// TIA Portal project "FillerMachine" (V15)
// Maquina llenadora Fuente Pura CCN

(* hardware
DEVICE "ET 200SP station_1"  ET 200SP-Station
   slot 0: "Rack_0"  Rack  6ES5 710-8MAx1
   slot 1: "PLC_1"  CPU 1510SP-1 PN  6ES7 510-1DJ01-0AB0  V2.5
   slot 2: "DI 8x24VDC ST_1"  DI 8x24VDC ST  6ES7 131-6BF00-0BA0  V1.1
      slot 1: "DI 8x24VDC ST_1"  DI 8x24VDC ST
   slot 3: "DI 8x24VDC ST_2"  DI 8x24VDC ST  6ES7 131-6BF01-0BA0  V0.0
      slot 1: "DI 8x24VDC ST_2"  DI 8x24VDC ST
   slot 4: "DI 8x24VDC ST_3"  DI 8x24VDC ST  6ES7 131-6BF01-0BA0  V0.0
      slot 1: "DI 8x24VDC ST_3"  DI 8x24VDC ST
   slot 5: "DQ 8x24VDC/0.5A ST_1"  DQ 8x24VDC/0.5A ST  6ES7 132-6BF01-0BA0  V0.0
      slot 1: "DQ 8x24VDC/0.5A ST_1"  DQ 8x24VDC/0.5A ST
   slot 6: "DQ 8x24VDC/0.5A ST_2"  DQ 8x24VDC/0.5A ST  6ES7 132-6BF01-0BA0  V0.0
      slot 1: "DQ 8x24VDC/0.5A ST_2"  DQ 8x24VDC/0.5A ST
   slot 7: "DQ 8x24VDC/0.5A ST_3"  DQ 8x24VDC/0.5A ST  6ES7 132-6BF01-0BA0  V0.0
      slot 1: "DQ 8x24VDC/0.5A ST_3"  DQ 8x24VDC/0.5A ST
   slot 8: "Server module_1"  Server module  6ES7 193-6PA00-0AA0  V1.1
      slot 1: "Server module_1"  Server module
   slot 127: "BA 2xRJ45"  BA 2xRJ45  6ES7 193-6AR00-0AA0  V0.0
      slot 32769: "Port_1"  6ES7 193-6AR00-0AA0
      slot 32770: "Port_2"  6ES7 193-6AR00-0AA0
DEVICE "HMI_1"  KTP600 Basic color PN
   slot 0: "HMI_1"  KTP600 Basic color PN  6AV6 647-0AD11-3AX0  12.0.0.0
   slot 1: "HMI_RT_2"  KTP600 Basic color PN  6AV6 647-0AD11-3AX0  12.0.0.0
   slot 5: "HMI_1.IE_CP_1"  PROFINET Interface  12.0.0.0
      slot 1: "PROFINET Interface_1"  PROFINET Interface
         slot 1: "Port_1"  Port
*)

// ===== PLC "PLC_1"  CPU 1510SP-1 PN =====

VAR_GLOBAL   // PLC tag table "Default tag table"
   "Stop_bitin" AT %I2.2 : Bool;
   "TriggerPump" AT %I0.1 : Bool;
   "ACKPump" AT %I0.2 : Bool;
   "TriggerClamp" AT %I0.3 : Bool;
   "ACKClamp" AT %I0.4 : Bool;
   "TriggerTransp1" AT %I0.5 : Bool;
   "ACKTransp1" AT %I0.6 : Bool;
   "TriggerTransp2" AT %I0.7 : Bool;
   "ACKTransp2" AT %I1.0 : Bool;
   "SensorTransIN2" AT %I1.1 : Bool;
   "SensorInBottle" AT %I1.2 : Bool;
   "SensorOutBottle" AT %I1.3 : Bool;
   "SensorLastBottle" AT %I1.4 : Bool;
   "SensorStageIN1" AT %I1.5 : Bool;
   "SensorLevelH" AT %I1.6 : Bool;
   "SensorLevelL" AT %I1.7 : Bool;
   "SensorBottleClamp" AT %I2.0 : Bool;
   "SensorTranspClamp" AT %I2.1 : Bool;
   "PumpVLow" AT %Q0.0 : Bool;
   "PumpVHigh" AT %Q0.1 : Bool;
   "PumpStop" AT %Q0.2 : Bool;
   "MotorTap" AT %Q0.3 : Bool;
   "MotorTrans1" AT %Q0.4 : Bool;
   "MotorTrans2" AT %Q0.5 : Bool;
   "EVPrincip" AT %Q0.6 : Bool;
   "EVBlowCylindIN" AT %Q0.7 : Bool;
   "EVCylindBottleHigh" AT %Q1.6 : Bool;
   "EVCylindNeck" AT %Q1.7 : Bool;
   "EVDoorIn" AT %Q2.2 : Bool;
   "EVDoorOut" AT %Q2.3 : Bool;
   "EVClampBotNeck" AT %Q2.4 : Bool;
   "EVClampDoor" AT %Q2.5 : Bool;
   "EVSuperClamp" AT %Q2.6 : Bool;
   "EVMandrilcylindUpDown" AT %Q2.7 : Bool;
   "MStartTouch" AT %M11.0 : Bool;
   "MBandaT-On" AT %M10.1 : Bool;
   "MFillScreen" AT %M10.2 : Bool;
   "MBottleProcess" AT %MD100 : DInt;
   "MBottleCounterIN" AT %MD4 : DInt;
   "MBottleCounterOut" AT %MD12 : DInt;
   "MEnableClampValve" AT %MD16 : DInt;
   "MFillFinish" AT %M10.3 : Bool;
   "M_stop_bit" AT %M11.1 : Bool;
   "F_TriggerPump" AT %M11.3 : Bool;
   "F_ACKPump" AT %M11.4 : Bool;
   "F_TriggerClamp" AT %M11.5 : Bool;
   "F_ACKClamp" AT %M11.6 : Bool;
   "F_TriggerTransp1" AT %M11.7 : Bool;
   "F_ACKTransp1" AT %M20.0 : Bool;
   "F_TriggerTransp2" AT %M20.1 : Bool;
   "F_ACKTransp2" AT %M20.2 : Bool;
   "SensorTransIN2_bit" AT %M20.3 : Bool;
   "SensorInBottle_bit" AT %M20.4 : Bool;
   "SensorOutBottle_bit" AT %M20.5 : Bool;
   "SensorLastBottle_bit" AT %M20.6 : Bool;
   "SensorStageIN1_bit" AT %M20.7 : Bool;
   "SensorLevelH_bit" AT %M21.0 : Bool;
   "SensorLevelL_bit" AT %M21.1 : Bool;
   "SensorBottleClamp_bit" AT %M21.2 : Bool;
   "SensorTranspClamp_bit" AT %M21.3 : Bool;
   "PumpVLow_bit" AT %M21.4 : Bool;
   "PumpVHigh_bit" AT %M21.5 : Bool;
   "PumpStop_bit" AT %M21.6 : Bool;
   "MotorTap_bit" AT %M21.7 : Bool;
   "MotorTrans1_bit" AT %M22.0 : Bool;
   "MotorTrans2_bit" AT %M22.1 : Bool;
   "EVPrincip_bit" AT %M22.2 : Bool;
   "EVBlowCylindIN_bit" AT %M22.3 : Bool;
   "EVMandrilcylindUpDown_bit" AT %M22.4 : Bool;
   "EVCylindNeck_bit" AT %M22.5 : Bool;
   "EVDoorIn_bit" AT %M22.6 : Bool;
   "EVDoorOut_bit" AT %M22.7 : Bool;
   "EVClampBotNeck_bit" AT %M23.0 : Bool;
   "EVClampDoor_bit" AT %M23.1 : Bool;
   "EVSuperClamp_bit" AT %M23.2 : Bool;
   "Alarm" AT %M24.0 : Bool;
   "F_TriggerPump_bit" AT %M24.1 : Bool;
   "F_ACKPump_bit" AT %M24.2 : Bool;
   "F_TriggerClamp_bit" AT %M24.3 : Bool;
   "F_ACKClamp_bit" AT %M24.4 : Bool;
   "F_TriggerTransp1_bit" AT %M24.5 : Bool;
   "F_ACKTransp1_bit" AT %M24.6 : Bool;
   "F_TriggerTransp2_bit" AT %M24.7 : Bool;
   "F_ACKTransp2_bit" AT %M25.0 : Bool;
   "Run" AT %M25.1 : Bool;
   "Stop_bit" AT %M25.2 : Bool;
   "StageLL0" AT %M25.3 : Bool;
   "StageLL1" AT %M25.4 : Bool;
   "MBottleCounterR" AT %M25.5 : Bool;
   "MBottleProcessR" AT %M25.6 : Bool;
   "StageLL2" AT %M25.7 : Bool;
   "MBottleclampRt" AT %M27.3 : Bool;
   "MBottleClamProcess" AT %MD101 : DInt;
   "MTrans1_touch" AT %M27.4 : Bool;
   "MTrans2_touch" AT %M27.5 : Bool;
   "MPump_touch" AT %M27.6 : Bool;
   "MClamp_touch" AT %M27.7 : Bool;
   "EVCylindBottleHigh_bit" AT %M28.0 : Bool;
   "StageLL3" AT %M28.1 : Bool;
   "StageLL4" AT %M28.2 : Bool;
   "StageLL5" AT %M28.3 : Bool;
   "StageLL6" AT %M28.4 : Bool;
   "StageLL7" AT %M28.5 : Bool;
   "StageLL8" AT %M28.6 : Bool;
   "StageLL9" AT %M28.7 : Bool;
   "StageLL10" AT %M29.0 : Bool;
   "StageLL11" AT %M29.1 : Bool;
   "Tag_1" AT %M400.1 : Bool;
   "StageLL12" AT %M29.2 : Bool;
   "StageLL13" AT %M29.3 : Bool;
   "StageLL14" AT %M29.4 : Bool;
   "Tag_2" AT %M400.2 : Bool;
   "StageLL00" AT %M29.5 : Bool;
   "MBottleCounterOutR" AT %M29.6 : Bool;
   "StageTap0" AT %M29.7 : Bool;
   "StageTap1" AT %M30.0 : Bool;
   "StageTap2" AT %M30.1 : Bool;
   "StageTap3" AT %M30.2 : Bool;
   "StageTap4" AT %M30.3 : Bool;
   "StageTap5" AT %M30.4 : Bool;
   "MTapProcessR" AT %M30.5 : Bool;
   "StageCon0" AT %M30.6 : Bool;
   "StageCon1" AT %M30.7 : Bool;
   "StageCon2" AT %M31.0 : Bool;
   "StageCon3" AT %M31.1 : Bool;
   "MConvT1R" AT %M31.2 : Bool;
   "MConvT2R" AT %M31.3 : Bool;
END_VAR

DATA_BLOCK "DB_Alarms"   // DB13
{ S7_Optimized_Access := 'FALSE' }
VERSION : 0.1
   VAR
      Stop_alm : Bool;
      T_Pump_alm : Bool;
      T_Transp1_alm : Bool;
      T_Transp2_alm : Bool;
      T_Clamp_alm_1 : Bool;
      alarms_active : Bool;
   END_VAR
BEGIN
END_DATA_BLOCK

// folder: System blocks/Program resources

DATA_BLOCK "IEC_Counter_0_DB"   // DB1
{ S7_Optimized_Access := 'TRUE' }
AUTHOR : Simatic
FAMILY : IEC
NAME : CNTR
VERSION : 1.0
// stored: InstanceOfName IEC_COUNTER
"IEC_COUNTER"
BEGIN
END_DATA_BLOCK

DATA_BLOCK "IEC_Timer_0_DB"   // DB2
{ S7_Optimized_Access := 'TRUE' }
AUTHOR : Simatic
FAMILY : IEC
NAME : IEC_TMR
VERSION : 1.0
// stored: InstanceOfName IEC_TIMER
"IEC_TIMER"
BEGIN
END_DATA_BLOCK

DATA_BLOCK "IEC_Timer_0_DB_1"   // DB3
{ S7_Optimized_Access := 'TRUE' }
AUTHOR : Simatic
FAMILY : IEC
NAME : IEC_TMR
VERSION : 1.0
// stored: InstanceOfName IEC_TIMER
"IEC_TIMER"
BEGIN
END_DATA_BLOCK

DATA_BLOCK "IEC_Timer_0_DB_2"   // DB5
{ S7_Optimized_Access := 'TRUE' }
AUTHOR : Simatic
FAMILY : IEC
NAME : IEC_TMR
VERSION : 1.0
// stored: InstanceOfName IEC_TIMER
"IEC_TIMER"
BEGIN
END_DATA_BLOCK

DATA_BLOCK "IEC_Timer_0_DB_4"   // DB6
{ S7_Optimized_Access := 'TRUE' }
AUTHOR : Simatic
FAMILY : IEC
NAME : IEC_TMR
VERSION : 1.0
// stored: InstanceOfName IEC_TIMER
"IEC_TIMER"
BEGIN
END_DATA_BLOCK

DATA_BLOCK "IEC_Timer_0_DB_5"   // DB7
{ S7_Optimized_Access := 'TRUE' }
AUTHOR : Simatic
FAMILY : IEC
NAME : IEC_TMR
VERSION : 1.0
// stored: InstanceOfName IEC_TIMER
"IEC_TIMER"
BEGIN
END_DATA_BLOCK

DATA_BLOCK "IEC_Timer_0_DB_17"   // DB8
{ S7_Optimized_Access := 'TRUE' }
AUTHOR : Simatic
FAMILY : IEC
NAME : IEC_TMR
VERSION : 1.0
// stored: InstanceOfName IEC_TIMER
"IEC_TIMER"
BEGIN
END_DATA_BLOCK

DATA_BLOCK "IEC_Timer_0_DB_7"   // DB9
{ S7_Optimized_Access := 'TRUE' }
AUTHOR : Simatic
FAMILY : IEC
NAME : IEC_TMR
VERSION : 1.0
// stored: InstanceOfName IEC_TIMER
"IEC_TIMER"
BEGIN
END_DATA_BLOCK

DATA_BLOCK "IEC_Timer_0_DB_8"   // DB10
{ S7_Optimized_Access := 'TRUE' }
AUTHOR : Simatic
FAMILY : IEC
NAME : IEC_TMR
VERSION : 1.0
// stored: InstanceOfName IEC_TIMER
"IEC_TIMER"
BEGIN
END_DATA_BLOCK

DATA_BLOCK "IEC_Timer_0_DB_9"   // DB11
{ S7_Optimized_Access := 'TRUE' }
AUTHOR : Simatic
FAMILY : IEC
NAME : IEC_TMR
VERSION : 1.0
// stored: InstanceOfName IEC_TIMER
"IEC_TIMER"
BEGIN
END_DATA_BLOCK

DATA_BLOCK "IEC_Timer_0_DB_10"   // DB12
{ S7_Optimized_Access := 'TRUE' }
AUTHOR : Simatic
FAMILY : IEC
NAME : IEC_TMR
VERSION : 1.0
// stored: InstanceOfName IEC_TIMER
"IEC_TIMER"
BEGIN
END_DATA_BLOCK

DATA_BLOCK "IEC_Counter_1_DB"   // DB14
{ S7_Optimized_Access := 'TRUE' }
AUTHOR : Simatic
FAMILY : IEC
NAME : CNTR
VERSION : 1.0
// stored: InstanceOfName IEC_COUNTER
"IEC_COUNTER"
BEGIN
END_DATA_BLOCK

DATA_BLOCK "IEC_Timer_0_DB_11"   // DB15
{ S7_Optimized_Access := 'TRUE' }
AUTHOR : Simatic
FAMILY : IEC
NAME : IEC_TMR
VERSION : 1.0
// stored: InstanceOfName IEC_TIMER
"IEC_TIMER"
BEGIN
END_DATA_BLOCK

DATA_BLOCK "IEC_Timer_0_DB_12"   // DB16
{ S7_Optimized_Access := 'TRUE' }
AUTHOR : Simatic
FAMILY : IEC
NAME : IEC_TMR
VERSION : 1.0
// stored: InstanceOfName IEC_TIMER
"IEC_TIMER"
BEGIN
END_DATA_BLOCK

DATA_BLOCK "IEC_Timer_0_DB_13"   // DB17
{ S7_Optimized_Access := 'TRUE' }
AUTHOR : Simatic
FAMILY : IEC
NAME : IEC_TMR
VERSION : 1.0
// stored: InstanceOfName IEC_TIMER
"IEC_TIMER"
BEGIN
END_DATA_BLOCK

DATA_BLOCK "IEC_Timer_0_DB_14"   // DB18
{ S7_Optimized_Access := 'TRUE' }
AUTHOR : Simatic
FAMILY : IEC
NAME : IEC_TMR
VERSION : 1.0
// stored: InstanceOfName IEC_TIMER
"IEC_TIMER"
BEGIN
END_DATA_BLOCK

DATA_BLOCK "IEC_Timer_0_DB_15"   // DB19
{ S7_Optimized_Access := 'TRUE' }
AUTHOR : Simatic
FAMILY : IEC
NAME : IEC_TMR
VERSION : 1.0
// stored: InstanceOfName IEC_TIMER
"IEC_TIMER"
BEGIN
END_DATA_BLOCK

DATA_BLOCK "IEC_Timer_0_DB_16"   // DB20
{ S7_Optimized_Access := 'TRUE' }
AUTHOR : Simatic
FAMILY : IEC
NAME : IEC_TMR
VERSION : 1.0
// stored: InstanceOfName IEC_TIMER
"IEC_TIMER"
BEGIN
END_DATA_BLOCK

// folder: (top level)

ORGANIZATION_BLOCK "Main"   // OB1, LAD, ProgramCycle
TITLE = "Main Program Sweep (Cycle)"
{ S7_Optimized_Access := 'TRUE' }
VERSION : 0.1
   VAR_INPUT
      Initial_Call : Bool;   // Initial call of this OB
      Remanence : Bool;   // =True, if remanent data are available
   END_VAR
   VAR_TEMP   // added for the SCL form of the ladder/FBD networks
      _w1 : Bool;
   END_VAR
BEGIN

REGION Network 1
   // Start  Stop Control
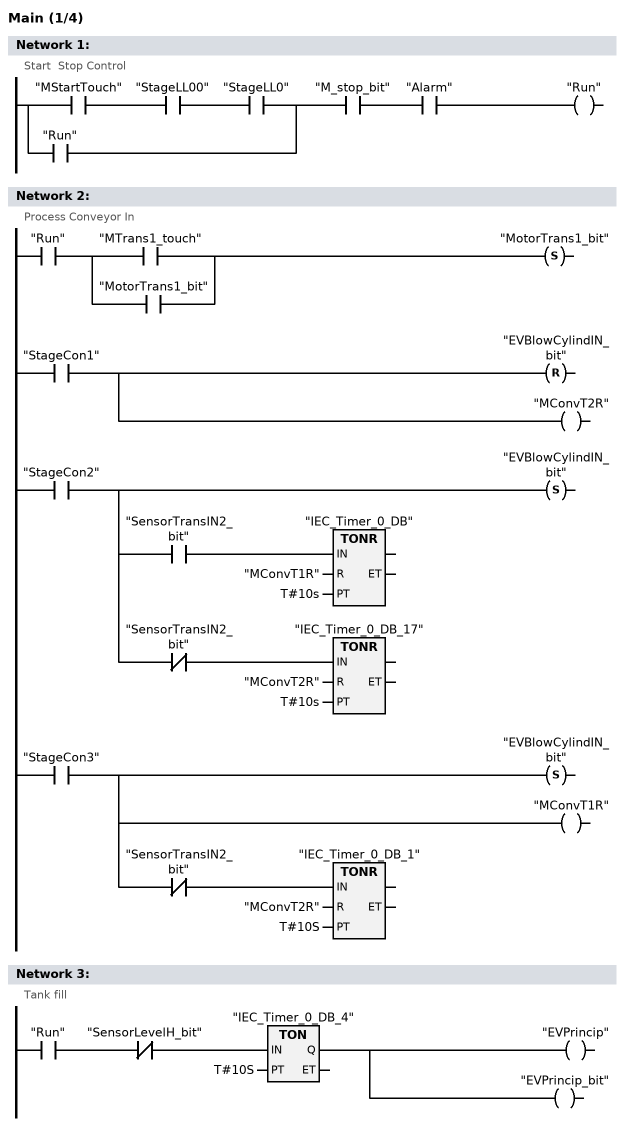
   RUNG wire#powerrail
      Contact( "MStartTouch" )
      Contact( "StageLL00" )
      Contact( "StageLL0" )
      wire#w1
      Contact( "M_stop_bit" )
      Contact( "Alarm" )
      Coil( "Run" )
   END_RUNG
   RUNG wire#powerrail
      Contact( "Run" )
   END_RUNG wire#w1
   // the same network as SCL:
   "Run" := (("MStartTouch" AND "StageLL00" AND "StageLL0") OR "Run") AND "M_stop_bit" AND "Alarm";
END_REGION

REGION Network 2
   // Process Conveyor In
   IF "Run" AND ("MTrans1_touch" OR "MotorTrans1_bit") THEN "MotorTrans1_bit" := TRUE; END_IF;
   IF "StageCon1" THEN "EVBlowCylindIN_bit" := FALSE; END_IF;
   "MConvT2R" := "StageCon1";
   IF "StageCon2" THEN "EVBlowCylindIN_bit" := TRUE; END_IF;
   "IEC_Timer_0_DB".TONR(IN := "StageCon2" AND "SensorTransIN2_bit", R := "MConvT1R", PT := T#10s);
   "IEC_Timer_0_DB_17".TONR(IN := "StageCon2" AND NOT "SensorTransIN2_bit", R := "MConvT2R", PT := T#10s);
   IF "StageCon3" THEN "EVBlowCylindIN_bit" := TRUE; END_IF;
   "MConvT1R" := "StageCon3";
   "IEC_Timer_0_DB_1".TONR(IN := "StageCon3" AND NOT "SensorTransIN2_bit", R := "MConvT2R", PT := T#10S);
END_REGION

REGION Network 3
   // Tank fill
   "IEC_Timer_0_DB_4".TON(IN := "Run" AND NOT "SensorLevelH_bit", PT := T#10S);
   "EVPrincip" := "IEC_Timer_0_DB_4".Q;
   "EVPrincip_bit" := "IEC_Timer_0_DB_4".Q;
END_REGION

REGION Network 4
   // Process Filling Bottle
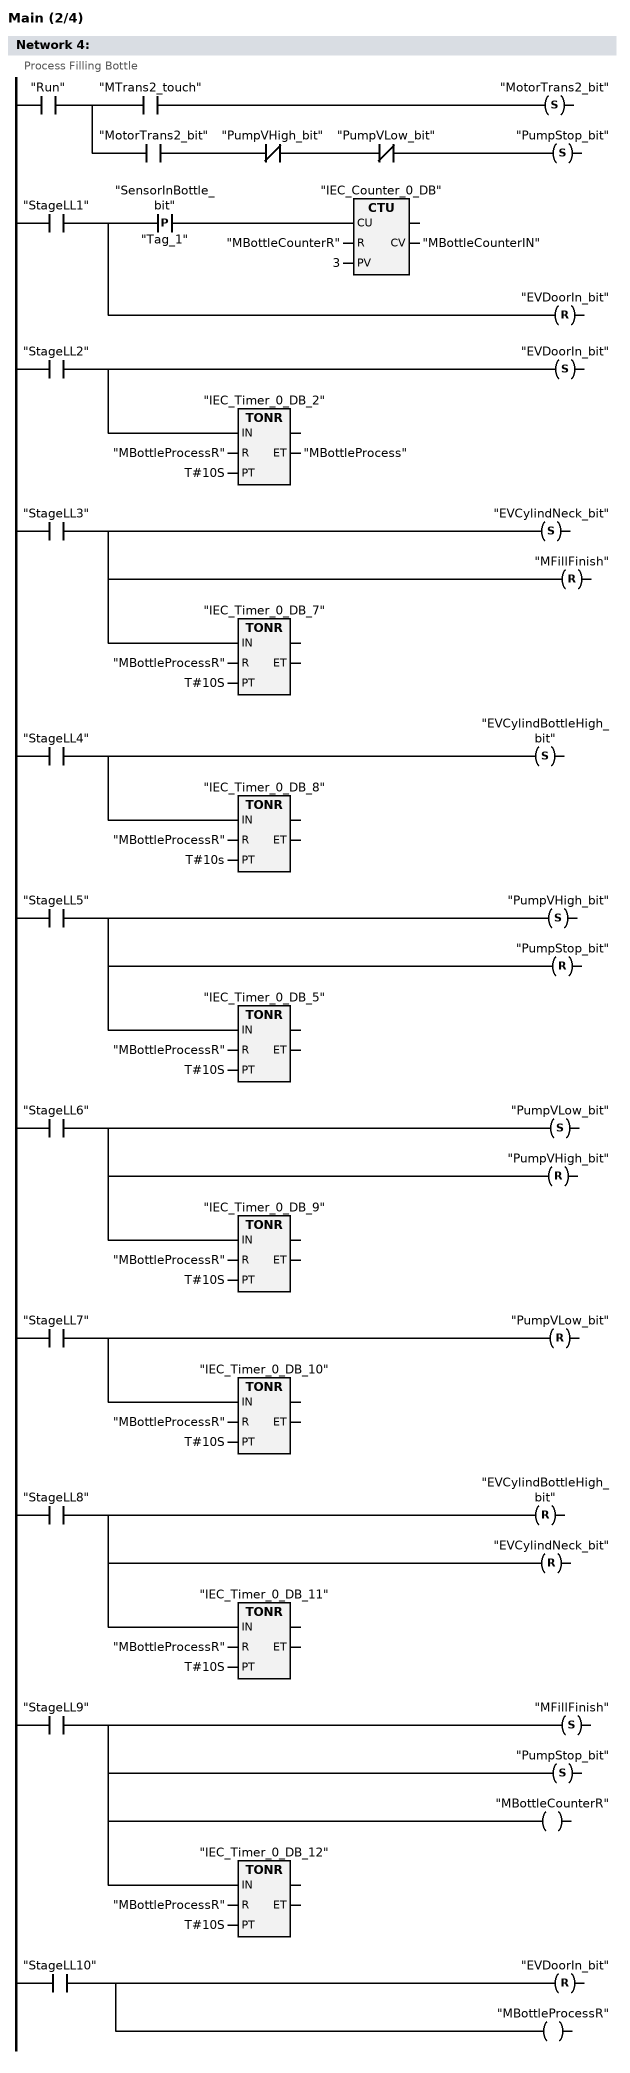
   IF "Run" AND "MTrans2_touch" THEN "MotorTrans2_bit" := TRUE; END_IF;
   IF "Run" AND "MotorTrans2_bit" AND NOT "PumpVHigh_bit" AND NOT "PumpVLow_bit" THEN
       "PumpStop_bit" := TRUE;
   END_IF;
   #_w1 := "StageLL1" AND "SensorInBottle_bit" AND NOT "Tag_1";   // rising edge of "SensorInBottle_bit"
   "Tag_1" := "SensorInBottle_bit";
   "IEC_Counter_0_DB".CTU(CU := #_w1, R := "MBottleCounterR", PV := 3, CV => "MBottleCounterIN");
   IF "StageLL1" THEN "EVDoorIn_bit" := FALSE; END_IF;
   IF "StageLL2" THEN "EVDoorIn_bit" := TRUE; END_IF;
   "IEC_Timer_0_DB_2".TONR(IN := "StageLL2", R := "MBottleProcessR", PT := T#10S, ET => "MBottleProcess");
   IF "StageLL3" THEN
       "EVCylindNeck_bit" := TRUE;
       "MFillFinish" := FALSE;
   END_IF;
   "IEC_Timer_0_DB_7".TONR(IN := "StageLL3", R := "MBottleProcessR", PT := T#10S);
   IF "StageLL4" THEN "EVCylindBottleHigh_bit" := TRUE; END_IF;
   "IEC_Timer_0_DB_8".TONR(IN := "StageLL4", R := "MBottleProcessR", PT := T#10s);
   IF "StageLL5" THEN
       "PumpVHigh_bit" := TRUE;
       "PumpStop_bit" := FALSE;
   END_IF;
   "IEC_Timer_0_DB_5".TONR(IN := "StageLL5", R := "MBottleProcessR", PT := T#10S);
   IF "StageLL6" THEN
       "PumpVLow_bit" := TRUE;
       "PumpVHigh_bit" := FALSE;
   END_IF;
   "IEC_Timer_0_DB_9".TONR(IN := "StageLL6", R := "MBottleProcessR", PT := T#10S);
   IF "StageLL7" THEN "PumpVLow_bit" := FALSE; END_IF;
   "IEC_Timer_0_DB_10".TONR(IN := "StageLL7", R := "MBottleProcessR", PT := T#10S);
   IF "StageLL8" THEN
       "EVCylindBottleHigh_bit" := FALSE;
       "EVCylindNeck_bit" := FALSE;
   END_IF;
   "IEC_Timer_0_DB_11".TONR(IN := "StageLL8", R := "MBottleProcessR", PT := T#10S);
   IF "StageLL9" THEN
       "MFillFinish" := TRUE;
       "PumpStop_bit" := TRUE;
   END_IF;
   "MBottleCounterR" := "StageLL9";
   "IEC_Timer_0_DB_12".TONR(IN := "StageLL9", R := "MBottleProcessR", PT := T#10S);
   IF "StageLL10" THEN "EVDoorIn_bit" := FALSE; END_IF;
   "MBottleProcessR" := "StageLL10";
END_REGION

REGION Network 5
   // Cylindre out
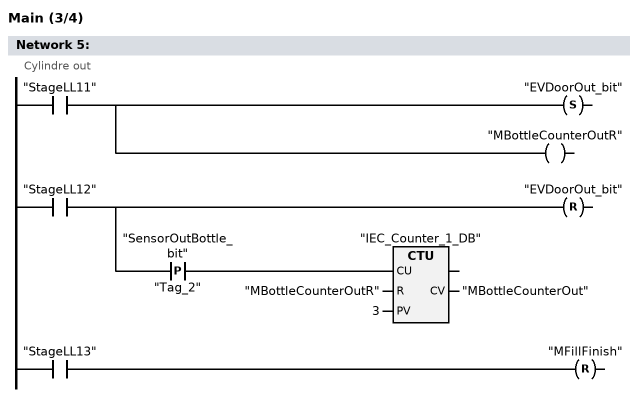
   IF "StageLL11" THEN "EVDoorOut_bit" := TRUE; END_IF;
   "MBottleCounterOutR" := "StageLL11";
   IF "StageLL12" THEN "EVDoorOut_bit" := FALSE; END_IF;
   #_w1 := "StageLL12" AND "SensorOutBottle_bit" AND NOT "Tag_2";   // rising edge of "SensorOutBottle_bit"
   "Tag_2" := "SensorOutBottle_bit";
   "IEC_Counter_1_DB".CTU(CU := #_w1, R := "MBottleCounterOutR", PV := 3, CV => "MBottleCounterOut");
   IF "StageLL13" THEN "MFillFinish" := FALSE; END_IF;
END_REGION

REGION Network 6
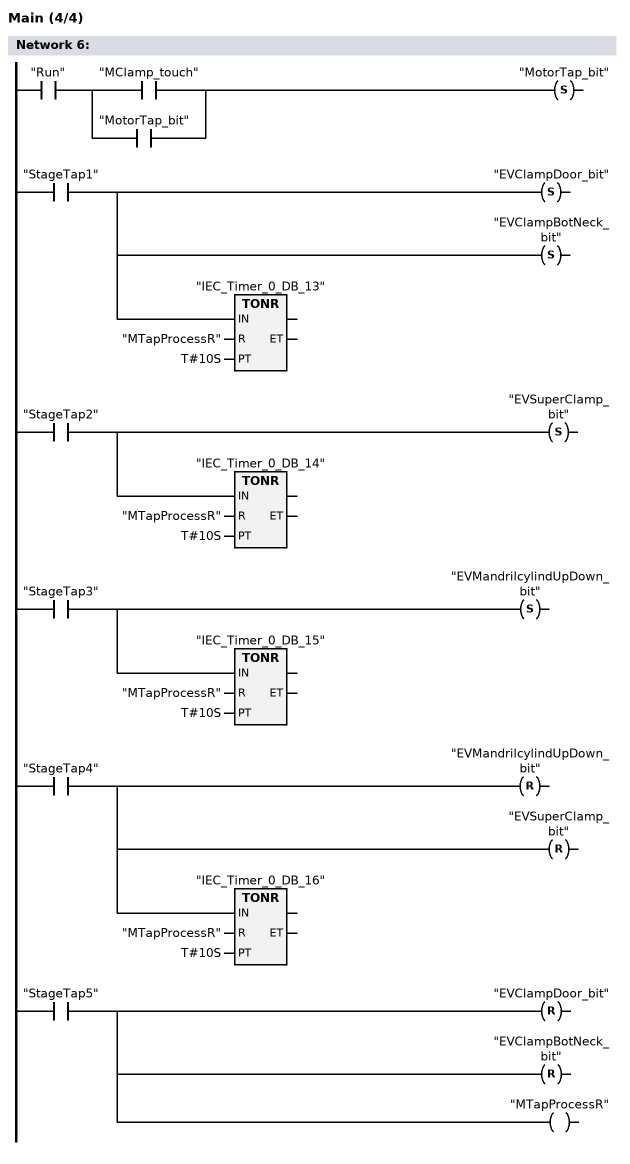
   IF "Run" AND ("MClamp_touch" OR "MotorTap_bit") THEN "MotorTap_bit" := TRUE; END_IF;
   IF "StageTap1" THEN
       "EVClampDoor_bit" := TRUE;
       "EVClampBotNeck_bit" := TRUE;
   END_IF;
   "IEC_Timer_0_DB_13".TONR(IN := "StageTap1", R := "MTapProcessR", PT := T#10S);
   IF "StageTap2" THEN "EVSuperClamp_bit" := TRUE; END_IF;
   "IEC_Timer_0_DB_14".TONR(IN := "StageTap2", R := "MTapProcessR", PT := T#10S);
   IF "StageTap3" THEN "EVMandrilcylindUpDown_bit" := TRUE; END_IF;
   "IEC_Timer_0_DB_15".TONR(IN := "StageTap3", R := "MTapProcessR", PT := T#10S);
   IF "StageTap4" THEN
       "EVMandrilcylindUpDown_bit" := FALSE;
       "EVSuperClamp_bit" := FALSE;
   END_IF;
   "IEC_Timer_0_DB_16".TONR(IN := "StageTap4", R := "MTapProcessR", PT := T#10S);
   IF "StageTap5" THEN
       "EVClampDoor_bit" := FALSE;
       "EVClampBotNeck_bit" := FALSE;
   END_IF;
   "MTapProcessR" := "StageTap5";
END_REGION

REGION Network 7
   // Minor bits
END_REGION
END_ORGANIZATION_BLOCK

ORGANIZATION_BLOCK "Alarms_block"   // OB123, LAD, ProgramCycle
TITLE = "Main Program Sweep (Cycle)"
{ S7_Optimized_Access := 'TRUE' }
VERSION : 0.1
   VAR_INPUT
      Initial_Call : Bool;   // Initial call of this OB
      Remanence : Bool;   // =True, if remanent data are available
   END_VAR
BEGIN

REGION Network 1
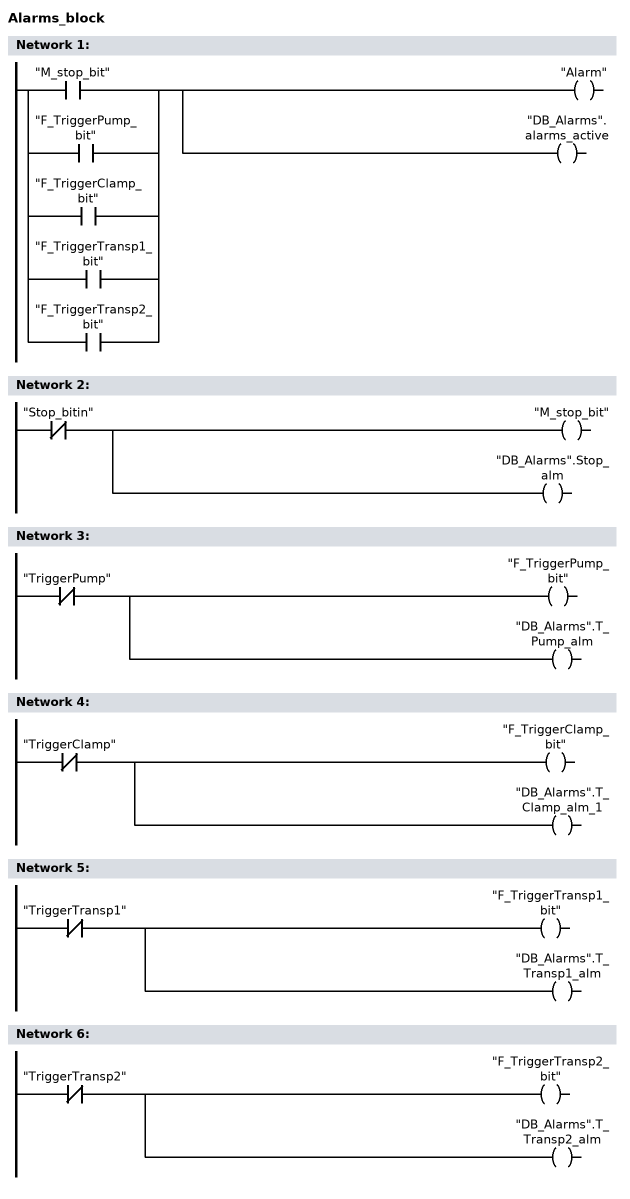
   RUNG wire#powerrail
      Contact( "M_stop_bit" )
      wire#w1
      Coil( "Alarm" )
   END_RUNG
   RUNG wire#powerrail
      Contact( "F_TriggerPump_bit" )
   END_RUNG wire#w1
   RUNG wire#powerrail
      Contact( "F_TriggerClamp_bit" )
   END_RUNG wire#w1
   RUNG wire#powerrail
      Contact( "F_TriggerTransp1_bit" )
   END_RUNG wire#w1
   RUNG wire#powerrail
      Contact( "F_TriggerTransp2_bit" )
   END_RUNG wire#w1
   RUNG wire#w1
      Coil( "DB_Alarms".alarms_active )
   END_RUNG
   // the same network as SCL:
   "Alarm" := "M_stop_bit" OR "F_TriggerPump_bit" OR "F_TriggerClamp_bit" OR "F_TriggerTransp1_bit" OR "F_TriggerTransp2_bit";
   "DB_Alarms".alarms_active := "Alarm";
END_REGION

REGION Network 2
   RUNG wire#powerrail
      I_Contact( "Stop_bitin" )
      wire#w1
      Coil( "M_stop_bit" )
   END_RUNG
   RUNG wire#w1
      Coil( "DB_Alarms".Stop_alm )
   END_RUNG
   // the same network as SCL:
   "M_stop_bit" := NOT "Stop_bitin";
   "DB_Alarms".Stop_alm := NOT "Stop_bitin";
END_REGION

REGION Network 3
   RUNG wire#powerrail
      I_Contact( "TriggerPump" )
      wire#w1
      Coil( "F_TriggerPump_bit" )
   END_RUNG
   RUNG wire#w1
      Coil( "DB_Alarms".T_Pump_alm )
   END_RUNG
   // the same network as SCL:
   "F_TriggerPump_bit" := NOT "TriggerPump";
   "DB_Alarms".T_Pump_alm := NOT "TriggerPump";
END_REGION

REGION Network 4
   RUNG wire#powerrail
      I_Contact( "TriggerClamp" )
      wire#w1
      Coil( "F_TriggerClamp_bit" )
   END_RUNG
   RUNG wire#w1
      Coil( "DB_Alarms".T_Clamp_alm_1 )
   END_RUNG
   // the same network as SCL:
   "F_TriggerClamp_bit" := NOT "TriggerClamp";
   "DB_Alarms".T_Clamp_alm_1 := NOT "TriggerClamp";
END_REGION

REGION Network 5
   RUNG wire#powerrail
      I_Contact( "TriggerTransp1" )
      wire#w1
      Coil( "F_TriggerTransp1_bit" )
   END_RUNG
   RUNG wire#w1
      Coil( "DB_Alarms".T_Transp1_alm )
   END_RUNG
   // the same network as SCL:
   "F_TriggerTransp1_bit" := NOT "TriggerTransp1";
   "DB_Alarms".T_Transp1_alm := NOT "TriggerTransp1";
END_REGION

REGION Network 6
   RUNG wire#powerrail
      I_Contact( "TriggerTransp2" )
      wire#w1
      Coil( "F_TriggerTransp2_bit" )
   END_RUNG
   RUNG wire#w1
      Coil( "DB_Alarms".T_Transp2_alm )
   END_RUNG
   // the same network as SCL:
   "F_TriggerTransp2_bit" := NOT "TriggerTransp2";
   "DB_Alarms".T_Transp2_alm := NOT "TriggerTransp2";
END_REGION
END_ORGANIZATION_BLOCK

ORGANIZATION_BLOCK "Stages"   // OB124, LAD, ProgramCycle
TITLE = "Main Program Sweep (Cycle)"
{ S7_Optimized_Access := 'TRUE' }
VERSION : 0.1
   VAR_INPUT
      Initial_Call : Bool;   // Initial call of this OB
      Remanence : Bool;   // =True, if remanent data are available
   END_VAR
   VAR_TEMP   // added for the SCL form of the ladder/FBD networks
      _w1 : Bool;
      _w2 : Bool;
   END_VAR
BEGIN

REGION Network 1
   // Stage0
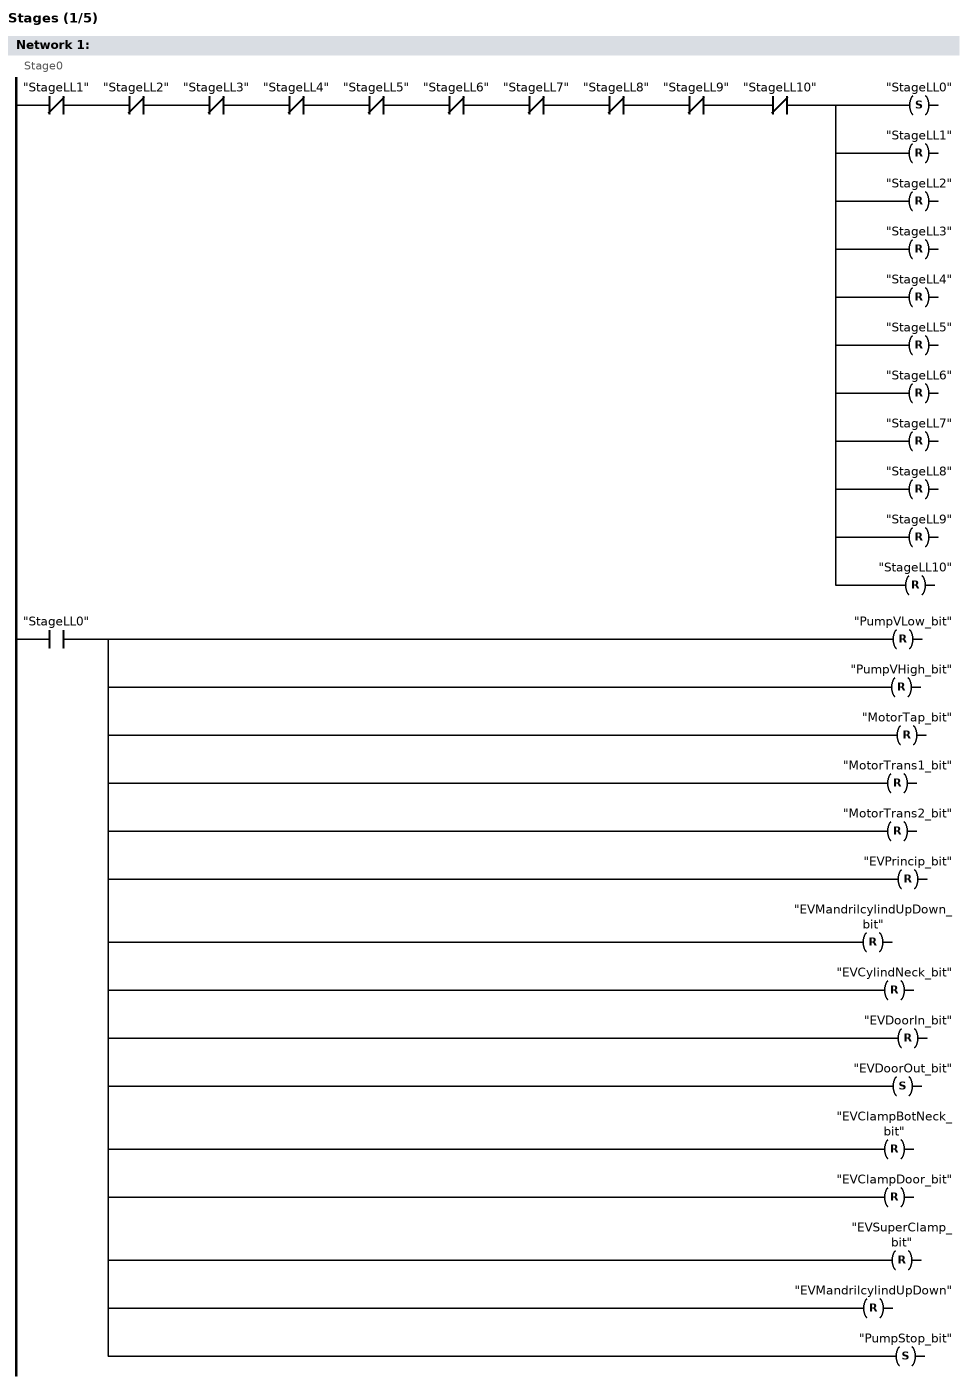
   RUNG wire#powerrail
      I_Contact( "StageLL1" )
      I_Contact( "StageLL2" )
      I_Contact( "StageLL3" )
      I_Contact( "StageLL4" )
      I_Contact( "StageLL5" )
      I_Contact( "StageLL6" )
      I_Contact( "StageLL7" )
      I_Contact( "StageLL8" )
      I_Contact( "StageLL9" )
      I_Contact( "StageLL10" )
      wire#w1
      S_Coil( "StageLL0" )
   END_RUNG
   RUNG wire#w1
      R_Coil( "StageLL1" )
   END_RUNG
   RUNG wire#w1
      R_Coil( "StageLL2" )
   END_RUNG
   RUNG wire#w1
      R_Coil( "StageLL3" )
   END_RUNG
   RUNG wire#w1
      R_Coil( "StageLL4" )
   END_RUNG
   RUNG wire#w1
      R_Coil( "StageLL5" )
   END_RUNG
   RUNG wire#w1
      R_Coil( "StageLL6" )
   END_RUNG
   RUNG wire#w1
      R_Coil( "StageLL7" )
   END_RUNG
   RUNG wire#w1
      R_Coil( "StageLL8" )
   END_RUNG
   RUNG wire#w1
      R_Coil( "StageLL9" )
   END_RUNG
   RUNG wire#w1
      R_Coil( "StageLL10" )
   END_RUNG
   RUNG wire#powerrail
      Contact( "StageLL0" )
      wire#w2
      R_Coil( "PumpVLow_bit" )
   END_RUNG
   RUNG wire#w2
      R_Coil( "PumpVHigh_bit" )
   END_RUNG
   RUNG wire#w2
      R_Coil( "MotorTap_bit" )
   END_RUNG
   RUNG wire#w2
      R_Coil( "MotorTrans1_bit" )
   END_RUNG
   RUNG wire#w2
      R_Coil( "MotorTrans2_bit" )
   END_RUNG
   RUNG wire#w2
      R_Coil( "EVPrincip_bit" )
   END_RUNG
   RUNG wire#w2
      R_Coil( "EVMandrilcylindUpDown_bit" )
   END_RUNG
   RUNG wire#w2
      R_Coil( "EVCylindNeck_bit" )
   END_RUNG
   RUNG wire#w2
      R_Coil( "EVDoorIn_bit" )
   END_RUNG
   RUNG wire#w2
      S_Coil( "EVDoorOut_bit" )
   END_RUNG
   RUNG wire#w2
      R_Coil( "EVClampBotNeck_bit" )
   END_RUNG
   RUNG wire#w2
      R_Coil( "EVClampDoor_bit" )
   END_RUNG
   RUNG wire#w2
      R_Coil( "EVSuperClamp_bit" )
   END_RUNG
   RUNG wire#w2
      R_Coil( "EVMandrilcylindUpDown" )
   END_RUNG
   RUNG wire#w2
      S_Coil( "PumpStop_bit" )
   END_RUNG
   // the same network as SCL:
   IF NOT "StageLL1" AND NOT "StageLL2" AND NOT "StageLL3" AND NOT "StageLL4" AND NOT "StageLL5" AND NOT "StageLL6" AND NOT "StageLL7" AND NOT "StageLL8" AND NOT "StageLL9" AND NOT "StageLL10" THEN
       "StageLL0" := TRUE;
   END_IF;
   #_w1 := NOT "StageLL1" AND NOT "StageLL2" AND NOT "StageLL3" AND NOT "StageLL4" AND NOT "StageLL5" AND NOT "StageLL6" AND NOT "StageLL7" AND NOT "StageLL8" AND NOT "StageLL9" AND NOT "StageLL10";
   IF #_w1 THEN
       "StageLL1" := FALSE;
       "StageLL2" := FALSE;
       "StageLL3" := FALSE;
       "StageLL4" := FALSE;
       "StageLL5" := FALSE;
       "StageLL6" := FALSE;
       "StageLL7" := FALSE;
       "StageLL8" := FALSE;
       "StageLL9" := FALSE;
       "StageLL10" := FALSE;
   END_IF;
   IF "StageLL0" THEN
       "PumpVLow_bit" := FALSE;
       "PumpVHigh_bit" := FALSE;
       "MotorTap_bit" := FALSE;
       "MotorTrans1_bit" := FALSE;
       "MotorTrans2_bit" := FALSE;
       "EVPrincip_bit" := FALSE;
       "EVMandrilcylindUpDown_bit" := FALSE;
       "EVCylindNeck_bit" := FALSE;
       "EVDoorIn_bit" := FALSE;
       "EVDoorOut_bit" := TRUE;
       "EVClampBotNeck_bit" := FALSE;
       "EVClampDoor_bit" := FALSE;
       "EVSuperClamp_bit" := FALSE;
       "EVMandrilcylindUpDown" := FALSE;
       "PumpStop_bit" := TRUE;
   END_IF;
END_REGION

REGION Network 2
   // Etapas de Cilindro de entrada y Llenado de Galones
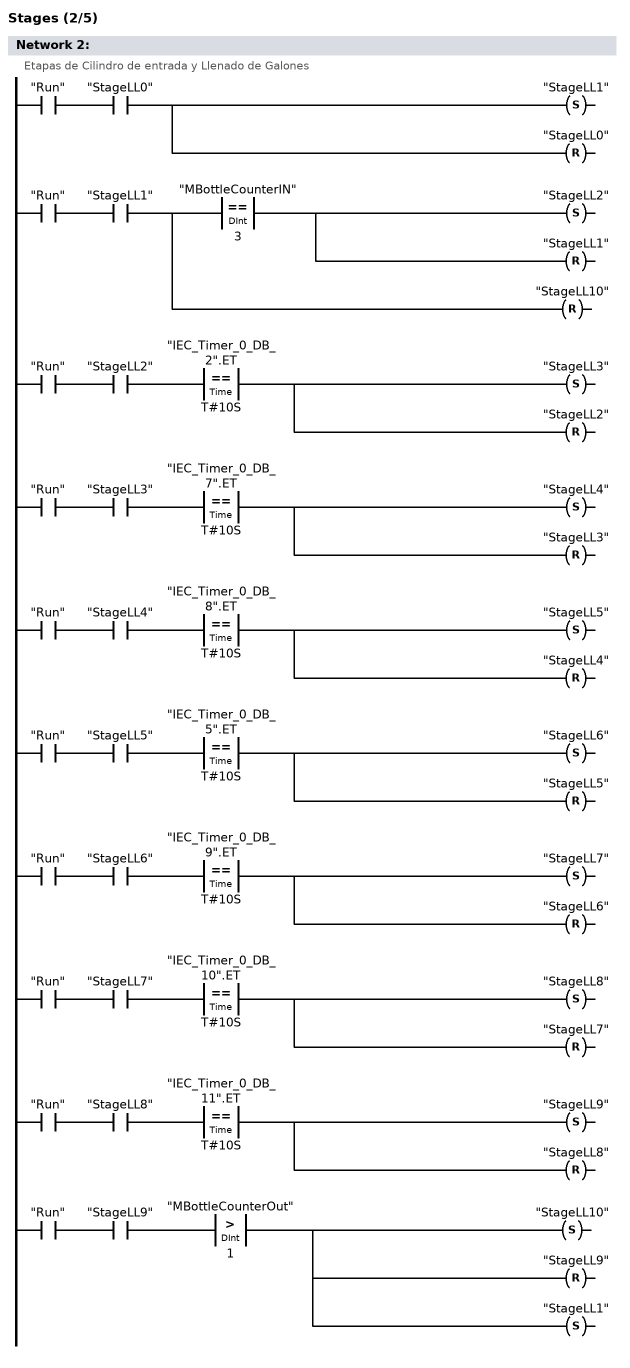
   RUNG wire#powerrail
      Contact( "Run" )
      Contact( "StageLL0" )
      wire#w1
      S_Coil( "StageLL1" )
   END_RUNG
   RUNG wire#w1
      R_Coil( "StageLL0" )
   END_RUNG
   RUNG wire#powerrail
      Contact( "Run" )
      Contact( "StageLL1" )
      wire#w2
      { S7_Templates := "SrcType := DInt" } EQ_Contact(in1 := "MBottleCounterIN", in2 := 3)
      wire#w3
      S_Coil( "StageLL2" )
   END_RUNG
   RUNG wire#w3
      R_Coil( "StageLL1" )
   END_RUNG
   RUNG wire#w2
      R_Coil( "StageLL10" )
   END_RUNG
   RUNG wire#powerrail
      Contact( "Run" )
      Contact( "StageLL2" )
      { S7_Templates := "SrcType := Time" } EQ_Contact(in1 := "IEC_Timer_0_DB_2".ET, in2 := T#10S)
      wire#w4
      S_Coil( "StageLL3" )
   END_RUNG
   RUNG wire#w4
      R_Coil( "StageLL2" )
   END_RUNG
   RUNG wire#powerrail
      Contact( "Run" )
      Contact( "StageLL3" )
      { S7_Templates := "SrcType := Time" } EQ_Contact(in1 := "IEC_Timer_0_DB_7".ET, in2 := T#10S)
      wire#w5
      S_Coil( "StageLL4" )
   END_RUNG
   RUNG wire#w5
      R_Coil( "StageLL3" )
   END_RUNG
   RUNG wire#powerrail
      Contact( "Run" )
      Contact( "StageLL4" )
      { S7_Templates := "SrcType := Time" } EQ_Contact(in1 := "IEC_Timer_0_DB_8".ET, in2 := T#10S)
      wire#w6
      S_Coil( "StageLL5" )
   END_RUNG
   RUNG wire#w6
      R_Coil( "StageLL4" )
   END_RUNG
   RUNG wire#powerrail
      Contact( "Run" )
      Contact( "StageLL5" )
      { S7_Templates := "SrcType := Time" } EQ_Contact(in1 := "IEC_Timer_0_DB_5".ET, in2 := T#10S)
      wire#w7
      S_Coil( "StageLL6" )
   END_RUNG
   RUNG wire#w7
      R_Coil( "StageLL5" )
   END_RUNG
   RUNG wire#powerrail
      Contact( "Run" )
      Contact( "StageLL6" )
      { S7_Templates := "SrcType := Time" } EQ_Contact(in1 := "IEC_Timer_0_DB_9".ET, in2 := T#10S)
      wire#w8
      S_Coil( "StageLL7" )
   END_RUNG
   RUNG wire#w8
      R_Coil( "StageLL6" )
   END_RUNG
   RUNG wire#powerrail
      Contact( "Run" )
      Contact( "StageLL7" )
      { S7_Templates := "SrcType := Time" } EQ_Contact(in1 := "IEC_Timer_0_DB_10".ET, in2 := T#10S)
      wire#w9
      S_Coil( "StageLL8" )
   END_RUNG
   RUNG wire#w9
      R_Coil( "StageLL7" )
   END_RUNG
   RUNG wire#powerrail
      Contact( "Run" )
      Contact( "StageLL8" )
      { S7_Templates := "SrcType := Time" } EQ_Contact(in1 := "IEC_Timer_0_DB_11".ET, in2 := T#10S)
      wire#w10
      S_Coil( "StageLL9" )
   END_RUNG
   RUNG wire#w10
      R_Coil( "StageLL8" )
   END_RUNG
   RUNG wire#powerrail
      Contact( "Run" )
      Contact( "StageLL9" )
      { S7_Templates := "SrcType := DInt" } GT_Contact(in1 := "MBottleCounterOut", in2 := 1)
      wire#w11
      S_Coil( "StageLL10" )
   END_RUNG
   RUNG wire#w11
      R_Coil( "StageLL9" )
   END_RUNG
   RUNG wire#w11
      S_Coil( "StageLL1" )
   END_RUNG
   // the same network as SCL:
   IF "Run" AND "StageLL0" THEN
       "StageLL1" := TRUE;
       "StageLL0" := FALSE;
   END_IF;
   #_w1 := "Run" AND "StageLL1";
   IF #_w1 AND ("MBottleCounterIN" = 3) THEN
       "StageLL2" := TRUE;
       "StageLL1" := FALSE;
   END_IF;
   IF #_w1 THEN "StageLL10" := FALSE; END_IF;
   IF "Run" AND "StageLL2" AND ("IEC_Timer_0_DB_2".ET = T#10S) THEN
       "StageLL3" := TRUE;
       "StageLL2" := FALSE;
   END_IF;
   IF "Run" AND "StageLL3" AND ("IEC_Timer_0_DB_7".ET = T#10S) THEN
       "StageLL4" := TRUE;
       "StageLL3" := FALSE;
   END_IF;
   IF "Run" AND "StageLL4" AND ("IEC_Timer_0_DB_8".ET = T#10S) THEN
       "StageLL5" := TRUE;
       "StageLL4" := FALSE;
   END_IF;
   IF "Run" AND "StageLL5" AND ("IEC_Timer_0_DB_5".ET = T#10S) THEN
       "StageLL6" := TRUE;
       "StageLL5" := FALSE;
   END_IF;
   IF "Run" AND "StageLL6" AND ("IEC_Timer_0_DB_9".ET = T#10S) THEN
       "StageLL7" := TRUE;
       "StageLL6" := FALSE;
   END_IF;
   IF "Run" AND "StageLL7" AND ("IEC_Timer_0_DB_10".ET = T#10S) THEN
       "StageLL8" := TRUE;
       "StageLL7" := FALSE;
   END_IF;
   IF "Run" AND "StageLL8" AND ("IEC_Timer_0_DB_11".ET = T#10S) THEN
       "StageLL9" := TRUE;
       "StageLL8" := FALSE;
   END_IF;
   IF "Run" AND "StageLL9" AND ("MBottleCounterOut" > 1) THEN "StageLL10" := TRUE; END_IF;
   #_w2 := "Run" AND "StageLL9" AND ("MBottleCounterOut" > 1);
   IF #_w2 THEN
       "StageLL9" := FALSE;
       "StageLL1" := TRUE;
   END_IF;
END_REGION

REGION Network 3
   // Etapas de Cilindro de Salida
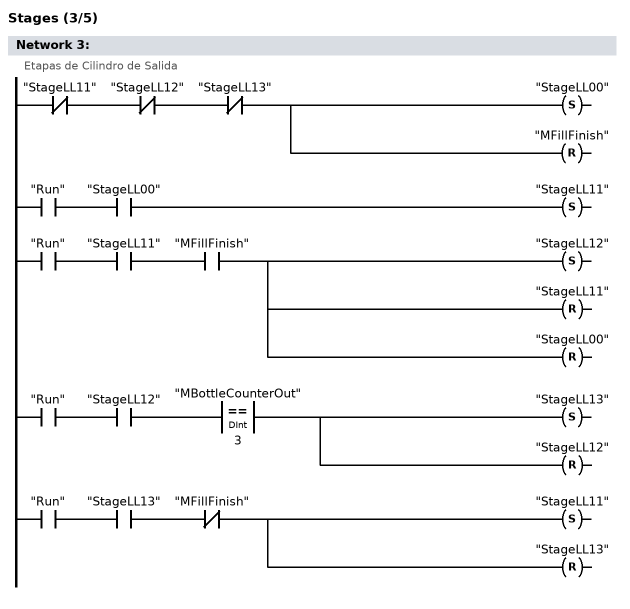
   RUNG wire#powerrail
      I_Contact( "StageLL11" )
      I_Contact( "StageLL12" )
      I_Contact( "StageLL13" )
      wire#w1
      S_Coil( "StageLL00" )
   END_RUNG
   RUNG wire#w1
      R_Coil( "MFillFinish" )
   END_RUNG
   RUNG wire#powerrail
      Contact( "Run" )
      Contact( "StageLL00" )
      S_Coil( "StageLL11" )
   END_RUNG
   RUNG wire#powerrail
      Contact( "Run" )
      Contact( "StageLL11" )
      Contact( "MFillFinish" )
      wire#w2
      S_Coil( "StageLL12" )
   END_RUNG
   RUNG wire#w2
      R_Coil( "StageLL11" )
   END_RUNG
   RUNG wire#w2
      R_Coil( "StageLL00" )
   END_RUNG
   RUNG wire#powerrail
      Contact( "Run" )
      Contact( "StageLL12" )
      { S7_Templates := "SrcType := DInt" } EQ_Contact(in1 := "MBottleCounterOut", in2 := 3)
      wire#w3
      S_Coil( "StageLL13" )
   END_RUNG
   RUNG wire#w3
      R_Coil( "StageLL12" )
   END_RUNG
   RUNG wire#powerrail
      Contact( "Run" )
      Contact( "StageLL13" )
      I_Contact( "MFillFinish" )
      wire#w4
      S_Coil( "StageLL11" )
   END_RUNG
   RUNG wire#w4
      R_Coil( "StageLL13" )
   END_RUNG
   // the same network as SCL:
   IF NOT "StageLL11" AND NOT "StageLL12" AND NOT "StageLL13" THEN
       "StageLL00" := TRUE;
       "MFillFinish" := FALSE;
   END_IF;
   IF "Run" AND "StageLL00" THEN "StageLL11" := TRUE; END_IF;
   IF "Run" AND "StageLL11" AND "MFillFinish" THEN "StageLL12" := TRUE; END_IF;
   #_w1 := "Run" AND "StageLL11" AND "MFillFinish";
   IF #_w1 THEN
       "StageLL11" := FALSE;
       "StageLL00" := FALSE;
   END_IF;
   IF "Run" AND "StageLL12" AND ("MBottleCounterOut" = 3) THEN
       "StageLL13" := TRUE;
       "StageLL12" := FALSE;
   END_IF;
   IF "Run" AND "StageLL13" AND NOT "MFillFinish" THEN
       "StageLL11" := TRUE;
       "StageLL13" := FALSE;
   END_IF;
END_REGION

REGION Network 4
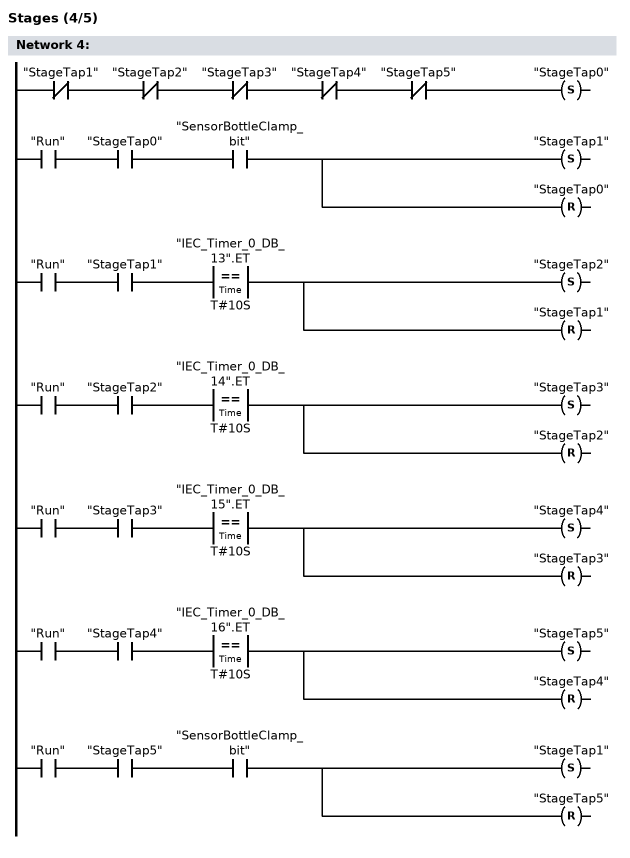
   RUNG wire#powerrail
      I_Contact( "StageTap1" )
      I_Contact( "StageTap2" )
      I_Contact( "StageTap3" )
      I_Contact( "StageTap4" )
      I_Contact( "StageTap5" )
      S_Coil( "StageTap0" )
   END_RUNG
   RUNG wire#powerrail
      Contact( "Run" )
      Contact( "StageTap0" )
      Contact( "SensorBottleClamp_bit" )
      wire#w1
      S_Coil( "StageTap1" )
   END_RUNG
   RUNG wire#w1
      R_Coil( "StageTap0" )
   END_RUNG
   RUNG wire#powerrail
      Contact( "Run" )
      Contact( "StageTap1" )
      { S7_Templates := "SrcType := Time" } EQ_Contact(in1 := "IEC_Timer_0_DB_13".ET, in2 := T#10S)
      wire#w2
      S_Coil( "StageTap2" )
   END_RUNG
   RUNG wire#w2
      R_Coil( "StageTap1" )
   END_RUNG
   RUNG wire#powerrail
      Contact( "Run" )
      Contact( "StageTap2" )
      { S7_Templates := "SrcType := Time" } EQ_Contact(in1 := "IEC_Timer_0_DB_14".ET, in2 := T#10S)
      wire#w3
      S_Coil( "StageTap3" )
   END_RUNG
   RUNG wire#w3
      R_Coil( "StageTap2" )
   END_RUNG
   RUNG wire#powerrail
      Contact( "Run" )
      Contact( "StageTap3" )
      { S7_Templates := "SrcType := Time" } EQ_Contact(in1 := "IEC_Timer_0_DB_15".ET, in2 := T#10S)
      wire#w4
      S_Coil( "StageTap4" )
   END_RUNG
   RUNG wire#w4
      R_Coil( "StageTap3" )
   END_RUNG
   RUNG wire#powerrail
      Contact( "Run" )
      Contact( "StageTap4" )
      { S7_Templates := "SrcType := Time" } EQ_Contact(in1 := "IEC_Timer_0_DB_16".ET, in2 := T#10S)
      wire#w5
      S_Coil( "StageTap5" )
   END_RUNG
   RUNG wire#w5
      R_Coil( "StageTap4" )
   END_RUNG
   RUNG wire#powerrail
      Contact( "Run" )
      Contact( "StageTap5" )
      Contact( "SensorBottleClamp_bit" )
      wire#w6
      S_Coil( "StageTap1" )
   END_RUNG
   RUNG wire#w6
      R_Coil( "StageTap5" )
   END_RUNG
   // the same network as SCL:
   IF NOT "StageTap1" AND NOT "StageTap2" AND NOT "StageTap3" AND NOT "StageTap4" AND NOT "StageTap5" THEN
       "StageTap0" := TRUE;
   END_IF;
   IF "Run" AND "StageTap0" AND "SensorBottleClamp_bit" THEN
       "StageTap1" := TRUE;
       "StageTap0" := FALSE;
   END_IF;
   IF "Run" AND "StageTap1" AND ("IEC_Timer_0_DB_13".ET = T#10S) THEN
       "StageTap2" := TRUE;
       "StageTap1" := FALSE;
   END_IF;
   IF "Run" AND "StageTap2" AND ("IEC_Timer_0_DB_14".ET = T#10S) THEN
       "StageTap3" := TRUE;
       "StageTap2" := FALSE;
   END_IF;
   IF "Run" AND "StageTap3" AND ("IEC_Timer_0_DB_15".ET = T#10S) THEN
       "StageTap4" := TRUE;
       "StageTap3" := FALSE;
   END_IF;
   IF "Run" AND "StageTap4" AND ("IEC_Timer_0_DB_16".ET = T#10S) THEN
       "StageTap5" := TRUE;
       "StageTap4" := FALSE;
   END_IF;
   IF "Run" AND "StageTap5" AND "SensorBottleClamp_bit" THEN
       "StageTap1" := TRUE;
       "StageTap5" := FALSE;
   END_IF;
END_REGION

REGION Network 5
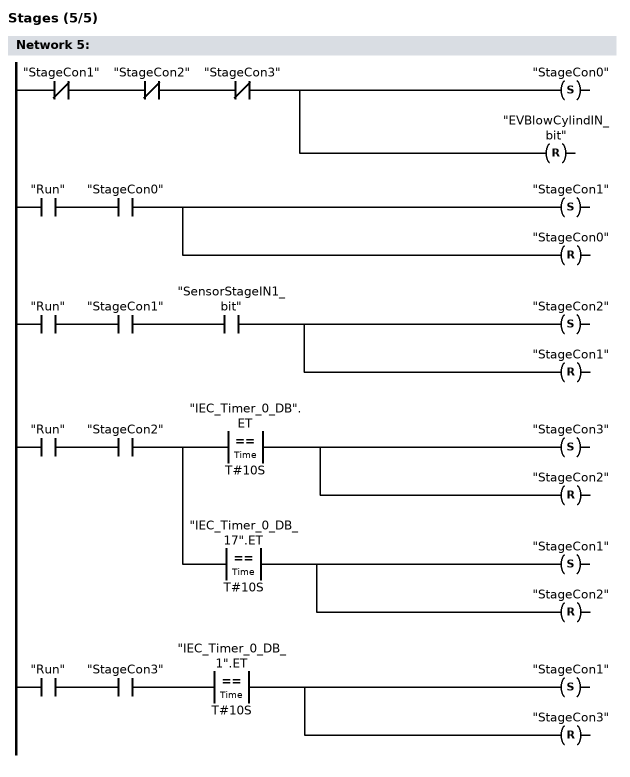
   RUNG wire#powerrail
      I_Contact( "StageCon1" )
      I_Contact( "StageCon2" )
      I_Contact( "StageCon3" )
      wire#w1
      S_Coil( "StageCon0" )
   END_RUNG
   RUNG wire#w1
      R_Coil( "EVBlowCylindIN_bit" )
   END_RUNG
   RUNG wire#powerrail
      Contact( "Run" )
      Contact( "StageCon0" )
      wire#w2
      S_Coil( "StageCon1" )
   END_RUNG
   RUNG wire#w2
      R_Coil( "StageCon0" )
   END_RUNG
   RUNG wire#powerrail
      Contact( "Run" )
      Contact( "StageCon1" )
      Contact( "SensorStageIN1_bit" )
      wire#w3
      S_Coil( "StageCon2" )
   END_RUNG
   RUNG wire#w3
      R_Coil( "StageCon1" )
   END_RUNG
   RUNG wire#powerrail
      Contact( "Run" )
      Contact( "StageCon2" )
      wire#w4
      { S7_Templates := "SrcType := Time" } EQ_Contact(in1 := "IEC_Timer_0_DB".ET, in2 := T#10S)
      wire#w5
      S_Coil( "StageCon3" )
   END_RUNG
   RUNG wire#w5
      R_Coil( "StageCon2" )
   END_RUNG
   RUNG wire#w4
      { S7_Templates := "SrcType := Time" } EQ_Contact(in1 := "IEC_Timer_0_DB_17".ET, in2 := T#10S)
      wire#w6
      S_Coil( "StageCon1" )
   END_RUNG
   RUNG wire#w6
      R_Coil( "StageCon2" )
   END_RUNG
   RUNG wire#powerrail
      Contact( "Run" )
      Contact( "StageCon3" )
      { S7_Templates := "SrcType := Time" } EQ_Contact(in1 := "IEC_Timer_0_DB_1".ET, in2 := T#10S)
      wire#w7
      S_Coil( "StageCon1" )
   END_RUNG
   RUNG wire#w7
      R_Coil( "StageCon3" )
   END_RUNG
   // the same network as SCL:
   IF NOT "StageCon1" AND NOT "StageCon2" AND NOT "StageCon3" THEN
       "StageCon0" := TRUE;
       "EVBlowCylindIN_bit" := FALSE;
   END_IF;
   IF "Run" AND "StageCon0" THEN
       "StageCon1" := TRUE;
       "StageCon0" := FALSE;
   END_IF;
   IF "Run" AND "StageCon1" AND "SensorStageIN1_bit" THEN
       "StageCon2" := TRUE;
       "StageCon1" := FALSE;
   END_IF;
   #_w1 := "Run" AND "StageCon2";
   IF #_w1 AND ("IEC_Timer_0_DB".ET = T#10S) THEN
       "StageCon3" := TRUE;
       "StageCon2" := FALSE;
   END_IF;
   IF #_w1 AND ("IEC_Timer_0_DB_17".ET = T#10S) THEN
       "StageCon1" := TRUE;
       "StageCon2" := FALSE;
   END_IF;
   IF "Run" AND "StageCon3" AND ("IEC_Timer_0_DB_1".ET = T#10S) THEN
       "StageCon1" := TRUE;
       "StageCon3" := FALSE;
   END_IF;
END_REGION
END_ORGANIZATION_BLOCK

ORGANIZATION_BLOCK "Minor_bits"   // OB125, LAD, ProgramCycle
TITLE = "Main Program Sweep (Cycle)"
{ S7_Optimized_Access := 'TRUE' }
VERSION : 0.1
   VAR_INPUT
      Initial_Call : Bool;   // Initial call of this OB
      Remanence : Bool;   // =True, if remanent data are available
   END_VAR
BEGIN

REGION Network 1
   // Minor Bits
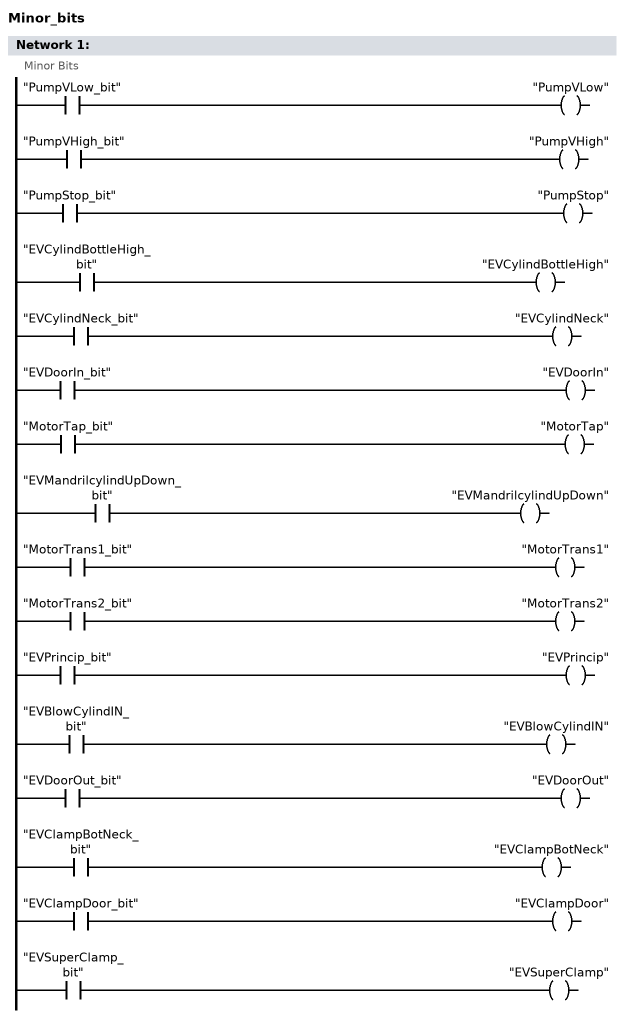
   RUNG wire#powerrail
      Contact( "PumpVLow_bit" )
      Coil( "PumpVLow" )
   END_RUNG
   RUNG wire#powerrail
      Contact( "PumpVHigh_bit" )
      Coil( "PumpVHigh" )
   END_RUNG
   RUNG wire#powerrail
      Contact( "PumpStop_bit" )
      Coil( "PumpStop" )
   END_RUNG
   RUNG wire#powerrail
      Contact( "EVCylindBottleHigh_bit" )
      Coil( "EVCylindBottleHigh" )
   END_RUNG
   RUNG wire#powerrail
      Contact( "EVCylindNeck_bit" )
      Coil( "EVCylindNeck" )
   END_RUNG
   RUNG wire#powerrail
      Contact( "EVDoorIn_bit" )
      Coil( "EVDoorIn" )
   END_RUNG
   RUNG wire#powerrail
      Contact( "MotorTap_bit" )
      Coil( "MotorTap" )
   END_RUNG
   RUNG wire#powerrail
      Contact( "EVMandrilcylindUpDown_bit" )
      Coil( "EVMandrilcylindUpDown" )
   END_RUNG
   RUNG wire#powerrail
      Contact( "MotorTrans1_bit" )
      Coil( "MotorTrans1" )
   END_RUNG
   RUNG wire#powerrail
      Contact( "MotorTrans2_bit" )
      Coil( "MotorTrans2" )
   END_RUNG
   RUNG wire#powerrail
      Contact( "EVPrincip_bit" )
      Coil( "EVPrincip" )
   END_RUNG
   RUNG wire#powerrail
      Contact( "EVBlowCylindIN_bit" )
      Coil( "EVBlowCylindIN" )
   END_RUNG
   RUNG wire#powerrail
      Contact( "EVDoorOut_bit" )
      Coil( "EVDoorOut" )
   END_RUNG
   RUNG wire#powerrail
      Contact( "EVClampBotNeck_bit" )
      Coil( "EVClampBotNeck" )
   END_RUNG
   RUNG wire#powerrail
      Contact( "EVClampDoor_bit" )
      Coil( "EVClampDoor" )
   END_RUNG
   RUNG wire#powerrail
      Contact( "EVSuperClamp_bit" )
      Coil( "EVSuperClamp" )
   END_RUNG
   // the same network as SCL:
   "PumpVLow" := "PumpVLow_bit";
   "PumpVHigh" := "PumpVHigh_bit";
   "PumpStop" := "PumpStop_bit";
   "EVCylindBottleHigh" := "EVCylindBottleHigh_bit";
   "EVCylindNeck" := "EVCylindNeck_bit";
   "EVDoorIn" := "EVDoorIn_bit";
   "MotorTap" := "MotorTap_bit";
   "EVMandrilcylindUpDown" := "EVMandrilcylindUpDown_bit";
   "MotorTrans1" := "MotorTrans1_bit";
   "MotorTrans2" := "MotorTrans2_bit";
   "EVPrincip" := "EVPrincip_bit";
   "EVBlowCylindIN" := "EVBlowCylindIN_bit";
   "EVDoorOut" := "EVDoorOut_bit";
   "EVClampBotNeck" := "EVClampBotNeck_bit";
   "EVClampDoor" := "EVClampDoor_bit";
   "EVSuperClamp" := "EVSuperClamp_bit";
END_REGION
END_ORGANIZATION_BLOCK

(* ===== HMI "HMI_RT_2" =====
system functions are stored by id; their names below are inferred from use
connection "HMI_Connection_1": ETHERNET, SMART_S7_1500_OMS

HMI tags "Default tag table"
   "HMI_Tag_1" : UInt AT %DB13.DBW0, 1 s
   "Tag_ScreenNumber" : UInt, internal
   "MStartTouch" : Bool = PLC MStartTouch AT %M11.0, 1 s
   "MTrans1_touch" : Bool = PLC MTrans1_touch AT %M27.4, 1 s
   "MTrans2_touch" : Bool = PLC MTrans2_touch AT %M27.5, 1 s
   "MClamp_touch" : Bool = PLC MClamp_touch AT %M27.7, 1 s

discrete alarms
   1: 'Alarma Paro de emergencia', class Errors, trigger "HMI_Tag_1" bit 0
   2: 'Disparo de Bomba', class Errors, trigger "HMI_Tag_1" bit 2
   3: 'Disparo del Motor Transportador 1', class Errors, trigger "HMI_Tag_1" bit 3
   4: 'Disparo del Motor Transportador 2', class Errors, trigger "HMI_Tag_1" bit 4
   5: 'Disparo del Motor Clamp', class Errors, trigger "HMI_Tag_1" bit 5
   6: 'Alarmas Activas', class Errors, trigger "HMI_Tag_1" bit 6

Template "Template_1" 320x240
   Button "Template_Button" at 266,202 size 52x37; TextOff 'Text'; PictureOff "ExitRuntime_KTP700_Basic_PN_TR"
      on Release: StopRuntime(0)
   Button "Template_Button_1" at 213,202 size 52x37; TextOff 'Text'
   Button "Template_Button_2" at 160,202 size 52x37; TextOff 'Text'
   Button "Template_Button_3" at 107,202 size 52x37; TextOff 'Text'; PictureOff "Graphic_3"
      on Release: ActivateScreen("Process", 0)
   Button "Template_Button_4" at 54,202 size 52x37; TextOff 'Text'; PictureOff "AlarmDisplay_KTP600_Basic_color_PN"
      on Release: ActivateScreen("Alarms", 0)
   Button "Alarms" at 1,202 size 52x37; TextOff 'Alarms'; PictureOn "AlarmDisplay_KTP600_Basic_color_PN"; PictureOff "Home"
      on Release: ActivateScreen("Main", 0)
   SymbolicIOField "Symbolic_IO_Field_Screen" at 69,7 size 164x24; TextOff '0'; TextOn '1'; TextList "TextList_ScreenNames"
      on Change: ActivateScreenByNumber("Tag_ScreenNumber", 0)
      ProcessValue <- "Tag_ScreenNumber"
   DateTimeField "HmiScreenItemData" at 235,19 size 85x19
   DateTimeField "HmiScreenItemData_1" at 235,0 size 85x19
   GraphicView "Logo" at 0,0 size 67x38; Picture "LogoHorizontal-e1441054646412"

screen "Main" 320x240, template "Template_1"
   on GenerateScreen: SetTag("Tag_ScreenNumber", 1)
   GraphicView "Graphic view_1" at 3,53 size 223x59; Picture "LogoHorizontal-e1441054646412"
   Button "Button_1" at 10,146 size 96x32; TextOff 'Start'
      on Press: SetBit("MStartTouch")

screen "Alarms" 320x240, template "Template_1"
   on GenerateScreen: SetTag("Tag_ScreenNumber", 2)
   AlarmView "Alarm view_1" at 0,40 size 320x141

screen "Process" 320x240, template "Template_1"
   on GenerateScreen: SetTag("Tag_ScreenNumber", 3)
   Button "Button_1" at 10,146 size 96x32; TextOff 'Bomba'
      on Press: SetBit("MStartTouch")
   Button "Button_2" at 10,102 size 96x32; TextOff 'B Trans 2'
      on Press: SetBit("MTrans2_touch")
   Button "Button_3" at 10,58 size 96x32; TextOff 'B Trans 1'
      on Press: SetBit("MTrans1_touch")
   Button "Button_4" at 124,58 size 96x32; TextOff 'Motor Tap.'
      on Press: SetBit("MClamp_touch")
*)